// TIA Portal V17 export
// export: Created 2025-06-25T13:13:31.4010412Z, ExportSetting WithDefaults, DisplayName Totally Integrated Automation Portal, DisplayVersion V17 Update 8, DisplayName TIA Portal Openness, DisplayVersion V17 Update 8, DisplayName TIA Portal Version Control Interface, DisplayVersion V17, DisplayName STEP 7 Professional, DisplayVersion V17 Update 8, DisplayName STEP 7 Safety, DisplayVersion V17 Update 6, DisplayName WinCC Advanced, DisplayVersion V17 Update 8
TYPE "stPIP_Regulator"
TITLE = Position-velocity controller
// Cascaded PI-P form
// stored: IsFailsafeCompliant false
   STRUCT
      bEnable : Bool;   // 1 = regulator on, 0 = regulator off
      fPV : Real;   // Process value (position)
      fPVvel : Real;   // Process value (velocity)
      fSP : Real;   // Setpoint (position)
      fOutMax : Real;   // Max regulator output
      fOutMin : Real;   // Min regulator output
      fVelMax : Real;   // Max velocity
      fVelMin : Real;   // Min velocity
      fOut : Real;   // Regulator output
      bManualMode : Bool;   // 1 = manual mode, 0 = auto
      fManualValue : Real;
      Kp : Real;   // Proportional gain (position)
      Tn : Real;   // Integral gain (reset time) (position)
      KpVel : Real;   // Proportional gain (velocity)
      TnVel : Real;   // Integral gain (velocity)
      fFeedbackHysteresis : Real;   // Deadband for velocity integrator
      bAtMin : Bool;   // Regulator output negative saturation
      bAtMax : Bool;   // Regulator output positive saturation
      bFault : Bool;   // 1 = regulator fault, 0 = ok
      nMode : USInt;   // 0 = Off, 1 = Auto, 2 = Manual
   END_STRUCT;
END_TYPE
